Yaskawa INFORM job: KRIS4(-224_-90).JBI

/JOB
//NAME KRIS4(-224_-90)
//POS
///NPOS 312,312,312,14,0,0
///TOOL 0
///POSTYPE PULSE
///PULSE
C00000=-126,-73357,-105376,18827,72039,77556
C00001=-35778,-73357,-105376,18827,72039,77556
C00002=-13505,189291,121101,6814,55937,83682
C00003=-119958,189291,121101,6814,55937,83682
C00004=-119958,189291,121101,6814,55937,83682
C00005=-119958,189291,121101,6814,104918,83682
C00006=-69507,150313,105301,6814,83622,83682
C00007=-72199,118597,79738,6814,89727,83682
C00008=14837,117754,79738,6814,55937,83682
C00009=44504,100666,44561,7265,69044,83737
C00010=106120,216,-72664,1265,72875,87293
C00011=133015,-103640,-65816,-3996,83698,82063
C00012=132086,-97485,-64003,-4135,58701,800
C00013=149065,-104779,-51399,7594,43822,5087
C00014=150289,-91952,-48932,6393,56924,6348
C00015=150393,-90903,-46944,6418,56235,6345
C00016=150312,-91064,-47459,6419,56476,6331
C00017=149346,-88536,-46306,6590,57139,6001
C00018=150281,-91600,-48374,6405,56765,6336
C00019=170298,-72142,-39060,11518,57888,13007
C00020=170167,-71928,-38964,11546,57956,12963
C00021=170167,-71173,-37488,11610,57441,12905
C00022=170167,-71393,-37919,11591,57591,12921
C00023=169145,-69698,-37147,11804,58123,12578
C00024=170288,-72356,-39514,11498,58052,13018
C00025=137447,-116054,-63762,19682,56909,-112
C00026=108026,-108792,-54867,-4103,57296,-6110
C00027=81416,-94598,-46445,-196,58741,-15925
C00028=81757,-93684,-45677,-246,58738,-15800
C00029=81757,-92858,-44382,-247,58365,-15799
C00030=81757,-93619,-45575,-246,58708,-15800
C00031=82768,-91970,-45027,-393,59221,-15429
C00032=81930,-94457,-46518,-272,58858,-15736
C00033=128580,-105651,-52299,-6719,58617,1362
C00034=130033,-102824,-49114,-6921,58227,1914
C00035=130033,-101283,-46878,-6964,57648,1951
C00036=130033,-101721,-47515,-6952,57813,1940
C00037=129738,-99854,-46987,-6872,58421,1793
C00038=130056,-102692,-48758,-6935,58079,1930
C00039=106734,-120076,-67764,-3834,59373,-6657
C00040=106734,-120076,-67764,-3834,76101,-81400
C00041=85493,-101158,-51309,-10056,72841,-87538
C00042=85426,-99920,-49312,-10091,72250,-87511
C00043=85426,-98477,-47146,-10119,71667,-87460
C00044=85426,-98764,-47576,-10113,71783,-87469
C00045=84550,-100156,-47986,-10204,71224,-87714
C00046=85920,-99324,-49419,-10033,72673,-87380
C00047=152431,-100504,-49770,-2471,77391,-65939
C00048=152805,-100536,-48996,-2423,76908,-65809
C00049=152805,-99353,-47240,-2427,76436,-65801
C00050=152805,-99697,-47754,-2425,76574,-65803
C00051=153892,-101565,-48290,-2277,75972,-65442
C00052=152767,-100966,-49728,-2425,77135,-65826
C00053=175766,-86349,-42944,18121,68088,-61743
C00054=175951,-86348,-42668,18137,67889,-61707
C00055=175951,-85124,-40623,18213,67291,-61803
C00056=175951,-85392,-41070,18196,67421,-61782
C00057=177474,-87024,-41664,18224,66648,-61355
C00058=175558,-86298,-43164,18103,68288,-61786
C00059=175558,-91829,-52585,17786,71106,-61349
C00060=197698,-109667,-58160,17366,61060,-54816
C00061=219000,-104945,-43712,24315,53908,-49637
C00062=231055,-104193,-38505,23952,48237,-46148
C00063=233659,-103437,-37306,23712,47268,-45306
C00064=233659,-102004,-35373,23879,46852,-45418
C00065=233659,-102412,-35924,23830,46971,-45386
C00066=237043,-102549,-35954,23321,46092,-44173
C00067=233629,-103481,-37368,23709,47288,-45313
C00068=215461,-127400,-43893,16870,58722,-48272
C00069=218544,-127186,-42626,17459,57581,-47480
C00070=218544,-125569,-40789,17514,57295,-47527
C00071=220330,-126171,-41362,17770,57042,-47002
C00072=227145,-126469,-41362,18757,55731,-45038
C00073=215464,-127169,-42828,16963,58209,-48354
C00074=177088,-126078,-40365,8704,67148,-58850
C00075=153631,-128510,-40310,2158,67069,-65285
C00076=154429,-128614,-40154,2389,66903,-65072
C00077=154429,-127009,-38360,2393,66624,-65076
C00078=154429,-127497,-38907,2392,66709,-65074
C00079=160472,-128938,-38826,4148,65740,-63473
C00080=156013,-128640,-39995,2844,66753,-64645
C00081=192579,-111155,-68057,11776,89768,-52211
C00082=192579,-150013,-128024,12422,106350,-50582
C00083=192579,-150013,-128024,12422,106350,-50582
C00084=146460,-104346,-58758,87,67702,-67205
C00085=142478,-76043,-30573,-21964,63223,-64301
C00086=140672,-66044,-21918,-20034,66227,-65754
C00087=140672,-65153,-20362,-20107,65757,-65668
C00088=140672,-65445,-20871,-20083,65909,-65696
C00089=141036,-66851,-21501,-20135,65677,-65523
C00090=140672,-66975,-23548,-19959,66721,-65841
C00091=152208,-64015,-24131,4423,60929,-65240
C00092=152310,-63243,-22366,4438,60237,-65228
C00093=152310,-62511,-21042,4457,59798,-65245
C00094=152310,-62815,-21590,4449,59978,-65238
C00095=152877,-64252,-22264,4382,59627,-65043
C00096=152310,-63427,-22700,4433,60345,-65224
C00097=165385,-47284,-4207,31110,46159,-66957
C00098=165600,-47601,-4286,31106,45987,-66914
C00099=165600,-46737,-2733,31361,45549,-67081
C00100=165600,-47131,-3441,31243,45749,-67005
C00101=166254,-48297,-4074,31163,45344,-66829
C00102=165393,-47522,-4616,31042,46268,-66913
C00103=159093,-40722,392,34170,55600,-67527
C00104=164207,-35275,5586,37104,52652,-66901
C00105=150105,-51391,-6646,37971,54466,-72302
C00106=160171,-66075,-30313,2176,67510,-69492
C00107=161226,-57856,-21857,1152,65004,-69036
C00108=161820,-56153,-18823,1098,63999,-68834
C00109=152948,-61625,-21548,2027,63029,-72005
C00110=152825,-64029,-24982,2024,63909,-72032
C00111=134056,-67322,-25852,-10196,66056,-78379
C00112=163216,-54448,-8591,-32623,76134,-65479
C00113=160229,-46098,-3230,-29804,80491,-68345
C00114=158451,-47284,-3883,-30173,79720,-68790
C00115=151927,-50958,-5849,-31450,76927,-70423
C00116=133676,-75568,-30882,-10874,62812,-78150
C00117=160835,-97860,-53381,-12033,68838,-69115
C00118=160835,-137865,-129483,-11388,94610,-71530
C00119=160835,-137865,-129483,-11388,94610,-71530
C00120=156474,-127565,-44757,2910,70220,-64434
C00121=182735,-127588,-36879,6458,67666,-54620
C00122=93853,-129558,-36709,-20996,60624,-77534
C00123=154263,-130476,-42112,-2655,69883,-62096
C00124=171605,-138664,-45039,640,62750,-56909
C00125=200673,-127969,-43722,7924,66337,-48717
C00126=199485,-124610,-40058,7659,65901,-49084
C00127=154854,-130863,-40060,-3943,63519,-61415
C00128=142889,-132361,-46546,-6897,66121,-64856
C00129=228263,-110324,-43358,23728,50162,-46686
C00130=234831,-107572,-40199,23168,48067,-44517
C00131=236443,-96869,-37709,21687,51363,-43058
C00132=226552,-115005,-54629,22549,54767,-46269
C00133=203481,-118873,-57487,18716,57337,-53342
C00134=208530,-112813,-51521,18479,55775,-51715
C00135=215259,-101474,-48621,17081,58299,-48731
C00136=205976,-112243,-55103,18172,58669,-52173
C00137=201958,-123065,-58725,3253,73839,-54936
C00138=197661,-129040,-56396,6313,64525,-57421
C00139=175928,-137233,-57000,3673,61831,-64313
C00140=171824,-140203,-61595,3068,63271,-65534
C00141=141766,-147898,-61645,-3344,56480,-74079
C00142=133776,-141760,-57056,-3252,60087,-76917
C00143=117425,-137681,-55374,-11246,62568,-80588
C00144=164064,-147455,-64185,-5609,61717,-65893
C00145=164064,-147455,-64185,-5609,61717,-65893
C00146=130860,-150279,-64151,6173,30547,11978
C00147=181055,-130986,-61566,-17152,51608,35195
C00148=182532,-124800,-57711,-17116,52650,35581
C00149=83593,-132502,-58869,6067,41588,-3855
C00150=101126,-133718,-57710,-9309,38222,6255
C00151=129711,-151516,-73375,-17379,42716,18129
C00152=134581,-137990,-74595,25751,56070,-1389
C00153=110654,-139179,-74777,26363,62443,-9081
C00154=121652,-127479,-66506,26214,60123,-5457
C00155=183969,-104449,-60936,13894,52742,18216
C00156=171621,-128341,-75090,18129,51623,12881
C00157=119711,-181360,-121572,24950,66300,-4723
C00158=119711,-181360,-121572,24950,66300,-4723
C00159=119711,-181360,-135603,24950,39029,-4723
C00160=119711,-181360,-135603,24950,39029,-4723
C00161=67118,-136665,-130676,31892,63753,5674
C00162=38158,-160025,-136084,39080,61805,7690
C00163=9060,-155984,-136090,36075,61852,27249
C00164=9060,-155984,-136090,36075,61852,27249
C00165=-35778,-73357,-105376,18827,72039,77556
C00166=-35778,-73357,-105376,18827,72039,77556
C00167=-121972,-60692,-66036,23906,48760,72917
C00168=-121972,-63565,-66036,13351,77444,72917
C00169=-114761,-44204,-50669,11461,76826,75375
C00170=-114807,-42889,-47501,11529,75582,75243
C00171=-114807,-42796,-46589,11554,75077,75195
C00172=-114807,-42822,-46844,11546,75217,75208
C00173=-114733,-44587,-47920,11539,74967,75210
C00174=-114807,-42889,-47501,11529,75582,75243
C00175=-106693,-40989,-47922,-8584,79047,76853
C00176=-106712,-40732,-46990,-8589,78608,76878
C00177=-106712,-40651,-45975,-8604,78031,76918
C00178=-106712,-40674,-46241,-8599,78181,76908
C00179=-106551,-42339,-47274,-8643,77981,76977
C00180=-106693,-40989,-47922,-8584,79047,76853
C00181=-119731,-42339,-42353,-28777,73600,71789
C00182=-120080,-41537,-40336,-28806,72749,71870
C00183=-120080,-41293,-39100,-28897,72189,72014
C00184=-120080,-41335,-39305,-28882,72281,71990
C00185=-120073,-43216,-40463,-28920,72059,72050
C00186=-120080,-41537,-40336,-28806,72749,71870
C00187=-101589,-42073,-44271,-32201,81327,76893
C00188=-104782,-94542,-85411,-8339,74693,77861
C00189=-98731,-154827,-131308,-9878,72678,80158
C00190=-98731,-154827,-131308,-9878,72678,80158
C00191=-98731,-154827,-131308,-9878,72678,80158
C00192=-141095,-137804,-121947,4358,90462,65341
C00193=-171917,-153174,-112370,-11397,78411,54227
C00194=-199110,-110397,-63847,-11158,69278,59316
C00195=-199661,-105459,-60576,-13729,71348,59282
C00196=-199661,-104714,-59434,-13753,71034,59321
C00197=-199661,-104881,-59692,-13747,71104,59313
C00198=-201697,-105978,-60019,-13785,70422,58683
C00199=-199661,-105459,-60576,-13729,71348,59282
C00200=-123960,-138876,-68675,-7989,69585,84604
C00201=-124072,-138705,-67366,-8043,68864,84619
C00202=-124072,-137612,-66165,-8049,68688,84634
C00203=-124072,-137824,-66399,-8047,68723,84632
C00204=-124282,-139731,-66590,-8126,67850,84627
C00205=-124072,-138655,-67314,-8040,68857,84622
C00206=-114984,-139242,-68510,12959,69151,83072
C00207=-114827,-138670,-67011,13034,68516,83052
C00208=-114827,-136931,-65095,13059,68238,83020
C00209=-114827,-137199,-65392,13055,68282,83025
C00210=-114467,-139013,-65570,13183,67430,83044
C00211=-114827,-138670,-67011,13034,68516,83052
C00212=-133085,-142772,-85485,9589,79895,78262
C00213=-119908,-107051,-70579,11526,87272,83253
C00214=-119905,-107270,-70562,11527,87152,83243
C00215=-119905,-106417,-69135,11528,86722,83203
C00216=-119905,-106577,-69401,11528,86804,83211
C00217=-119887,-108279,-69933,11533,86265,83166
C00218=-119905,-107341,-70681,11527,87191,83247
C00219=-147950,-101609,-70952,-8097,88078,75282
C00220=-148936,-101577,-69519,-8210,87121,75014
C00221=-148936,-100979,-68423,-8210,86757,75037
C00222=-148936,-101159,-68752,-8210,86867,75032
C00223=-149395,-102566,-69230,-8263,86398,74908
C00224=-148936,-101830,-69986,-8210,87277,75005
C00225=-165354,-89650,-65481,-16319,85072,70011
C00226=-165779,-89873,-64407,-16347,84242,69973
C00227=-165779,-89214,-62991,-16359,83730,70041
C00228=-165779,-89312,-63202,-16357,83805,70031
C00229=-166355,-90439,-63644,-16386,83393,69883
C00230=-165632,-89756,-64683,-16338,84492,69992
C00231=-143601,-106428,-78314,-14904,88558,77172
C00232=-127839,-150907,-89343,-18520,59767,2936
C00233=-132953,-138286,-79588,-18019,59168,1112
C00234=-137115,-133470,-77672,-17386,59565,-529
C00235=-137115,-131953,-75830,-17447,59223,-475
C00236=-137115,-132842,-76915,-17411,59423,-507
C00237=-136304,-129881,-76308,-17304,60683,-404
C00238=-137115,-133253,-77414,-17394,59515,-521
C00239=-181699,-110020,-71549,-8619,60587,-17610
C00240=-181630,-109868,-71398,-8637,60579,-17583
C00241=-181630,-109061,-70095,-8670,60195,-17555
C00242=-181630,-109567,-70911,-8650,60436,-17574
C00243=-179495,-107200,-70173,-9064,61418,-16842
C00244=-181374,-109783,-71626,-8682,60786,-17501
C00245=-138549,-156108,-92608,-17680,56945,-638
C00246=-92857,-152389,-93170,1138,51221,11865
C00247=-89241,-137374,-84375,135,53495,13313
C00248=-89241,-137236,-84209,135,53464,13313
C00249=-89241,-136248,-83020,135,53240,13313
C00250=-89241,-136629,-83479,135,53327,13313
C00251=-90422,-134246,-82978,442,54247,12852
C00252=-88987,-137859,-84464,69,53301,13413
C00253=-151501,-140988,-86034,14129,58291,-10466
C00254=-150678,-138310,-84494,13941,58574,-10114
C00255=-150678,-137164,-83136,13977,58332,-10146
C00256=-150678,-137515,-83554,13966,58407,-10136
C00257=-149186,-134345,-82896,13563,59357,-9449
C00258=-151128,-139683,-85226,14047,58399,-10308
C00259=-154150,-131986,-81973,14219,60800,-11137
C00260=-88152,-132772,-82145,-148,54492,13740
C00261=-103700,-131599,-81415,11358,56317,183
C00262=-119170,-146244,-89248,14851,56054,-5885
C00263=-129919,-160370,-92966,-12704,53201,3154
C00264=-134642,-143084,-81504,-11683,54346,1201
C00265=-146256,-142714,-76617,-8488,45375,-2851
C00266=-190967,-116324,-69611,1501,49612,-20855
C00267=-164928,-143381,-78407,-9170,42235,-9240
C00268=-155273,-152427,-83467,-13136,41921,-4825
C00269=-158141,-110882,-79211,-11782,79402,69500
C00270=-156021,-110302,-75029,-11867,77473,70419
C00271=-164693,-106825,-70970,-11824,75528,67599
C00272=-175106,-97531,-67666,-11410,76738,63853
C00273=-131080,-121620,-80305,-3109,79327,78003
C00274=-136811,-120114,-75832,127,77816,75713
C00275=-120666,-121905,-76299,1170,77058,81080
C00276=-118816,-123903,-80121,1281,78355,81709
C00277=-109990,-123163,-79929,1817,78452,84652
C00278=-122003,-121691,-75603,8260,77024,79739
C00279=-127593,-119006,-72089,19029,78419,76519
C00280=-135969,-121502,-76764,18008,81762,74135
C00281=-157702,-146234,-81795,15058,76702,66164
C00282=-157352,-138799,-66788,13808,73912,66272
C00283=-167304,-136290,-63149,11542,74320,63270
C00284=-135907,-141176,-63619,18589,67249,72053
C00285=-148278,-138995,-66659,15795,72315,68901
C00286=-146781,-141799,-67483,-9190,63470,73790
C00287=-172222,-135689,-66769,-11071,63352,65466
C00288=-167439,-135845,-70174,-10586,65898,66819
C00289=-192902,-115042,-63146,-20265,60680,60371
C00290=-199703,-112368,-59358,-19763,58226,58217
C00291=-207207,-100813,-56084,-18051,60307,54942
C00292=-170801,-131743,-76226,-21430,65470,67743
C00293=-164740,-137810,-91614,-20635,72894,68588
C00294=-164740,-137810,-91614,-20635,72894,68588
C00295=-149447,-191890,-120181,-21381,67024,75156
C00296=-149584,-192173,-120256,-21405,66899,75131
C00297=-149584,-192173,-120256,-21405,66899,75131
C00298=-114761,-44204,-50669,11461,76826,75375
C00299=-117144,-39713,-45211,12000,78898,74743
C00300=-110396,-38535,-44464,10422,78117,77015
C00301=-114060,-50823,-52718,11111,71580,75110
C00302=-124826,-51246,-53710,-3634,72889,70409
C00303=-126627,-37483,-45033,-3511,81308,69522
C00304=-133904,-35632,-43787,-1986,81245,67064
C00305=-133954,-36259,-45628,-1970,82055,67034
C00306=-135284,-28260,-32637,-27547,76219,65313
C00307=-136156,-27594,-30758,-27439,75206,65218
C00308=-139816,-25285,-26607,-31214,71734,64504
C00309=-131832,-52683,-49405,-33204,65462,69826
C00310=-109380,-75662,-60137,-33198,63885,64520
C00311=-9054,-143647,-113334,5954,77551,79151
BC00000=192652,674564,1075172
BC00001=85490,674564,1075172
BC00002=85490,674564,1075172
BC00003=388274,674564,1075172
BC00004=388274,1057170,1075172
BC00005=388274,1057170,1075172
BC00006=266797,1098418,1075172
BC00007=245359,1165153,1075172
BC00008=171901,1306919,981729
BC00009=145084,1358673,1075172
BC00010=282424,1358673,1075172
BC00011=324887,1177345,1075172
BC00012=324887,1177345,1033512
BC00013=324887,1177345,1033512
BC00014=324887,1177345,1033512
BC00015=324887,1177345,1033512
BC00016=324887,1177345,1033512
BC00017=324887,1177345,1033512
BC00018=324887,1177345,1033512
BC00019=324887,1177345,1033512
BC00020=324887,1177345,1033512
BC00021=324887,1177345,1033512
BC00022=324887,1177345,1033512
BC00023=324887,1177345,1033512
BC00024=324887,1177345,1033512
BC00025=324887,1177345,1033512
BC00026=324887,1177345,1033512
BC00027=324887,1177345,1033512
BC00028=324887,1177345,1033512
BC00029=324887,1177345,1033512
BC00030=324887,1177345,1033512
BC00031=324887,1177345,1033512
BC00032=324887,1177345,1033512
BC00033=324887,1177345,1033512
BC00034=324887,1177345,1033512
BC00035=324887,1177345,1033512
BC00036=324887,1177345,1033512
BC00037=324887,1177345,1033512
BC00038=324887,1177345,1033512
BC00039=324887,1177345,1033512
BC00040=324887,1147445,1033512
BC00041=324887,1147445,1033512
BC00042=324887,1147445,1033512
BC00043=324887,1147445,1033512
BC00044=324887,1147445,1033512
BC00045=324887,1147445,1033512
BC00046=324887,1147445,1033512
BC00047=324887,1147445,1033512
BC00048=324887,1147445,1033512
BC00049=324887,1147445,1033512
BC00050=324887,1147445,1033512
BC00051=324887,1147445,1033512
BC00052=324887,1147445,1033512
BC00053=324887,1147445,1033512
BC00054=324887,1147445,1033512
BC00055=324887,1147445,1033512
BC00056=324887,1147445,1033512
BC00057=324887,1147445,1033512
BC00058=324887,1147445,1033512
BC00059=324887,1147445,1033512
BC00060=324887,1147445,1033512
BC00061=324887,1119707,1033512
BC00062=324887,1119707,1033512
BC00063=324887,1119707,1033512
BC00064=324887,1119707,1033512
BC00065=324887,1119707,1033512
BC00066=324887,1119707,1033512
BC00067=324887,1119707,1033512
BC00068=324887,1119707,1033512
BC00069=324887,1119707,1033512
BC00070=324887,1119707,1033512
BC00071=324887,1119707,1033512
BC00072=324887,1119707,1033512
BC00073=324887,1119707,1033512
BC00074=346918,1122350,1033512
BC00075=365620,1122350,1033512
BC00076=365620,1122350,1033512
BC00077=365620,1122350,1033512
BC00078=365620,1122350,1033512
BC00079=365620,1122350,1033512
BC00080=365620,1122350,1033512
BC00081=365620,1122350,1033512
BC00082=365620,1122350,1033512
BC00083=365620,1290426,1033512
BC00084=365620,1290426,1028316
BC00085=365620,1290426,1028316
BC00086=365620,1290426,1028316
BC00087=365620,1290426,1028316
BC00088=365620,1290426,1028316
BC00089=365620,1290426,1028316
BC00090=365620,1290426,1028316
BC00091=365620,1290426,1028316
BC00092=365620,1290426,1028316
BC00093=365620,1290426,1028316
BC00094=365620,1290426,1028316
BC00095=365620,1290426,1028316
BC00096=365620,1290426,1028316
BC00097=365620,1290426,1028316
BC00098=365620,1290426,1028316
BC00099=365620,1290426,1028316
BC00100=365620,1290426,1028316
BC00101=365620,1290426,1028316
BC00102=365620,1290426,1028316
BC00103=365620,1290426,1028316
BC00104=365620,1290426,1028316
BC00105=365620,1290426,1028316
BC00106=365620,1290426,1028316
BC00107=365620,1290426,1028316
BC00108=365620,1290426,1028316
BC00109=365620,1290426,1028316
BC00110=365620,1290426,1028316
BC00111=365620,1290426,1028316
BC00112=365620,1290426,1028316
BC00113=365620,1290426,1028316
BC00114=365620,1290426,1028316
BC00115=365620,1290426,1028316
BC00116=365620,1290426,1028316
BC00117=365620,1290426,1028316
BC00118=365620,1290426,1028316
BC00119=365620,1203984,1028316
BC00120=365620,1122350,1033512
BC00121=354696,1118911,1033512
BC00122=354696,1118911,1033512
BC00123=354696,1118911,1033512
BC00124=289412,1118911,1033512
BC00125=299099,1130329,1033512
BC00126=299099,1130329,1033512
BC00127=299099,1130329,1033512
BC00128=299099,1130329,1033512
BC00129=323037,1120469,1018827
BC00130=323037,1120469,1018827
BC00131=323037,1120469,1018827
BC00132=323037,1120469,1018827
BC00133=323037,1103765,1018827
BC00134=323037,1103765,1018827
BC00135=323037,1103765,1018827
BC00136=323037,1103765,1018827
BC00137=323037,1103765,1018827
BC00138=323037,1103765,1018827
BC00139=323037,1103765,1018827
BC00140=323037,1103765,1018827
BC00141=359327,1103765,1018827
BC00142=359327,1103765,1018827
BC00143=359327,1103765,1018827
BC00144=359327,1103765,1018827
BC00145=320666,1103765,1061735
BC00146=320666,1151385,1061735
BC00147=348115,1151385,988526
BC00148=348115,1151385,988526
BC00149=348115,1151385,988526
BC00150=348115,1151385,988526
BC00151=348115,1151385,988526
BC00152=348115,1151385,988526
BC00153=317563,1137817,963781
BC00154=317563,1137817,963781
BC00155=317563,1137817,963781
BC00156=317563,1137817,963781
BC00157=317563,1137817,963781
BC00158=357256,1203577,1061822
BC00159=340361,1234496,1068927
BC00160=340361,1313599,1068927
BC00161=331783,1191875,1070117
BC00162=326822,1083331,1070805
BC00163=344400,890386,1072234
BC00164=344400,743708,1072234
BC00165=295326,674564,1075172
BC00166=295326,676593,1075172
BC00167=295326,676846,813323
BC00168=336009,760791,731248
BC00169=336009,760791,731248
BC00170=336009,760791,731248
BC00171=336009,760791,731248
BC00172=336009,760791,731248
BC00173=336009,760791,731248
BC00174=336009,760791,731248
BC00175=292309,760791,731248
BC00176=292309,760791,731248
BC00177=292309,760791,731248
BC00178=292309,760791,731248
BC00179=292309,760791,731248
BC00180=292309,760791,731248
BC00181=292309,760791,731248
BC00182=292309,760791,731248
BC00183=292309,760791,731248
BC00184=292309,760791,731248
BC00185=292309,760791,731248
BC00186=292309,760791,731248
BC00187=292309,760791,731248
BC00188=292309,760791,731248
BC00189=292309,760791,979870
BC00190=314389,897937,979870
BC00191=314389,914237,695700
BC00192=349616,923854,695700
BC00193=349616,946341,695700
BC00194=318497,960445,891334
BC00195=318497,960445,891334
BC00196=318497,960445,891334
BC00197=318497,960445,891334
BC00198=318497,960445,891334
BC00199=318497,960445,891334
BC00200=318497,960445,891334
BC00201=318497,960445,891334
BC00202=318497,960445,891334
BC00203=318497,960445,891334
BC00204=318497,960445,891334
BC00205=318497,960445,891334
BC00206=348006,960445,891333
BC00207=348006,960445,891333
BC00208=348006,960445,891333
BC00209=348006,960445,891333
BC00210=348006,960445,891333
BC00211=348006,960445,891333
BC00212=348006,960445,891333
BC00213=348006,960445,891333
BC00214=348006,960445,891333
BC00215=348006,960445,891333
BC00216=348006,960445,891333
BC00217=348006,960445,891333
BC00218=348006,960445,891333
BC00219=348006,960445,891333
BC00220=348006,960445,891333
BC00221=348006,960445,891333
BC00222=348006,960445,891333
BC00223=348006,960445,891333
BC00224=348006,960445,891333
BC00225=317395,960445,891333
BC00226=317395,960445,891333
BC00227=317395,960445,891333
BC00228=317395,960445,891333
BC00229=317395,960445,891333
BC00230=317395,960445,891333
BC00231=317395,960445,891333
BC00232=317395,960445,891333
BC00233=317395,960445,891333
BC00234=317395,960445,891333
BC00235=317395,960445,891333
BC00236=317395,960445,891333
BC00237=317395,960445,891333
BC00238=317395,960445,891333
BC00239=317395,960445,891333
BC00240=317395,960445,891333
BC00241=317395,960445,891333
BC00242=317395,960445,891333
BC00243=317395,960445,891333
BC00244=317395,960445,891333
BC00245=317395,960445,891333
BC00246=339742,960445,891333
BC00247=339741,960446,891330
BC00248=339741,960446,891330
BC00249=339741,960446,891330
BC00250=339741,960446,891330
BC00251=339741,960446,891330
BC00252=339741,960446,891330
BC00253=339741,960446,891330
BC00254=339741,960446,891330
BC00255=339741,960446,891330
BC00256=339741,960446,891330
BC00257=339741,960446,891330
BC00258=339741,960446,891330
BC00259=339741,960446,891330
BC00260=339741,960446,891330
BC00261=339741,960446,891330
BC00262=339741,960446,891330
BC00263=310327,960446,891330
BC00264=310327,960446,891330
BC00265=310327,960446,891330
BC00266=310327,960446,891330
BC00267=310327,960446,891330
BC00268=310327,960446,891330
BC00269=310327,960446,891330
BC00270=310327,960446,891330
BC00271=310327,960446,891330
BC00272=310327,960446,891330
BC00273=310327,960446,891330
BC00274=310327,960446,891330
BC00275=310327,960446,891326
BC00276=310327,960446,891326
BC00277=351201,960446,891326
BC00278=351201,960446,891326
BC00279=351201,960446,891326
BC00280=351201,960446,891326
BC00281=351201,960446,891326
BC00282=351201,960446,891326
BC00283=351201,960446,891326
BC00284=351201,960446,891326
BC00285=351201,960446,891326
BC00286=335367,960446,891326
BC00287=335367,960446,891326
BC00288=335367,960446,891326
BC00289=335367,960446,891326
BC00290=335367,960446,891326
BC00291=335367,960446,891326
BC00292=335367,960446,891326
BC00293=335367,960446,891326
BC00294=352748,960446,1069813
BC00295=352748,960446,1069813
BC00296=352748,842200,1069813
BC00297=352748,842200,743331
BC00298=336009,760791,731248
BC00299=336010,760791,731247
BC00300=336010,760792,731244
BC00301=336010,760791,731247
BC00302=336010,760791,731247
BC00303=336010,760791,731247
BC00304=336010,760791,731247
BC00305=336010,760791,731247
BC00306=336010,760791,731247
BC00307=336010,760791,731247
BC00308=336010,760791,731247
BC00309=336010,760791,731247
BC00310=361481,703019,979319
BC00311=361481,673970,979319
EC00000=-1986524,-556476
EC00001=-1986524,-556476
EC00002=-1986524,-556476
EC00003=-1986524,-556476
EC00004=-1986524,-556476
EC00005=-1986524,-556476
EC00006=-1986524,-556476
EC00007=-1986524,-556476
EC00008=-1986524,-556476
EC00009=-1986524,-556476
EC00010=-1986524,-556476
EC00011=-1986524,-556476
EC00012=-1986524,-556476
EC00013=-1986524,-556476
EC00014=-1986524,-556476
EC00015=-1986524,-556476
EC00016=-1986524,-556476
EC00017=-1986524,-556476
EC00018=-1986524,-556476
EC00019=-1986524,-556476
EC00020=-1986524,-556476
EC00021=-1986524,-556476
EC00022=-1986524,-556476
EC00023=-1986524,-556476
EC00024=-1986524,-556476
EC00025=-1986524,-556476
EC00026=-1986524,-556476
EC00027=-1986524,-556476
EC00028=-1986524,-556476
EC00029=-1986524,-556476
EC00030=-1986524,-556476
EC00031=-1986524,-556476
EC00032=-1986524,-556476
EC00033=-1986524,-556476
EC00034=-1986524,-556476
EC00035=-1986524,-556476
EC00036=-1986524,-556476
EC00037=-1986524,-556476
EC00038=-1986524,-556476
EC00039=-1986524,-556476
EC00040=-1986524,-556476
EC00041=-1986524,-556476
EC00042=-1986524,-556476
EC00043=-1986524,-556476
EC00044=-1986524,-556476
EC00045=-1986524,-556476
EC00046=-1986524,-556476
EC00047=-1986524,-556476
EC00048=-1986524,-556476
EC00049=-1986524,-556476
EC00050=-1986524,-556476
EC00051=-1986524,-556476
EC00052=-1986524,-556476
EC00053=-1986524,-556476
EC00054=-1986524,-556476
EC00055=-1986524,-556476
EC00056=-1986524,-556476
EC00057=-1986524,-556476
EC00058=-1986524,-556476
EC00059=-1986524,-556476
EC00060=-1986524,-556476
EC00061=-1986524,-556476
EC00062=-1986524,-556476
EC00063=-1986524,-556476
EC00064=-1986524,-556476
EC00065=-1986524,-556476
EC00066=-1986524,-556476
EC00067=-1986524,-556476
EC00068=-1986524,-556476
EC00069=-1986524,-556476
EC00070=-1986524,-556476
EC00071=-1986524,-556476
EC00072=-1986524,-556476
EC00073=-1986524,-556476
EC00074=-1986524,-556476
EC00075=-1986524,-556476
EC00076=-1986524,-556476
EC00077=-1986524,-556476
EC00078=-1986524,-556476
EC00079=-1986524,-556476
EC00080=-1986524,-556476
EC00081=-1986524,-556476
EC00082=-1986524,-556476
EC00083=-1986524,-556476
EC00084=-1986525,-556476
EC00085=-1986525,-556476
EC00086=-1986525,-556476
EC00087=-1986525,-556476
EC00088=-1986525,-556476
EC00089=-1986525,-556476
EC00090=-1986525,-556476
EC00091=-1986525,-556476
EC00092=-1986525,-556476
EC00093=-1986525,-556476
EC00094=-1986525,-556476
EC00095=-1986525,-556476
EC00096=-1986525,-556476
EC00097=-1986525,-556476
EC00098=-1986525,-556476
EC00099=-1986525,-556476
EC00100=-1986525,-556476
EC00101=-1986525,-556476
EC00102=-1986525,-556476
EC00103=-1986525,-556476
EC00104=-1986525,-556476
EC00105=-1986525,-556476
EC00106=-1986525,-556476
EC00107=-1986525,-556476
EC00108=-1986525,-556476
EC00109=-1986525,-556476
EC00110=-1986525,-556476
EC00111=-1986525,-556476
EC00112=-1986525,-556476
EC00113=-1986525,-556476
EC00114=-1986525,-556476
EC00115=-1986525,-556476
EC00116=-1986525,-556476
EC00117=-1986525,-556476
EC00118=-1986525,-556476
EC00119=-1986525,-556476
EC00120=-1986524,-556476
EC00121=-1986524,-556476
EC00122=-1986524,-556476
EC00123=-1986524,-556476
EC00124=-1986524,-556476
EC00125=-1986524,-556476
EC00126=-1986524,-556476
EC00127=-1986524,-556476
EC00128=-1986524,-556476
EC00129=-1986524,-556476
EC00130=-1986524,-556476
EC00131=-1986524,-556476
EC00132=-1986524,-556476
EC00133=-1986524,-556476
EC00134=-1986524,-556476
EC00135=-1986524,-556476
EC00136=-1986524,-556476
EC00137=-1986524,-556476
EC00138=-1986524,-556476
EC00139=-1986524,-556476
EC00140=-1986524,-556476
EC00141=-1986524,-556476
EC00142=-1986524,-556476
EC00143=-1986524,-556476
EC00144=-1986524,-556476
EC00145=-1986524,-556476
EC00146=-1986524,-556476
EC00147=-1986524,-556476
EC00148=-1986524,-556476
EC00149=-1986524,-556476
EC00150=-1986524,-556476
EC00151=-1986524,-556476
EC00152=-1986524,-556476
EC00153=-1986524,-556476
EC00154=-1986524,-556476
EC00155=-1986524,-556476
EC00156=-1986524,-556476
EC00157=-1986524,-556476
EC00158=-1986524,-556476
EC00159=-1986524,-556476
EC00160=-1986524,-556476
EC00161=-1924386,-453661
EC00162=-1888448,-394196
EC00163=-1813786,-270658
EC00164=-1813786,-270658
EC00165=-1660311,-16712
EC00166=-1178646,554555
EC00167=-1144025,556476
EC00168=-1144025,556476
EC00169=-1144025,556476
EC00170=-1144025,556476
EC00171=-1144025,556476
EC00172=-1144025,556476
EC00173=-1144025,556476
EC00174=-1144025,556476
EC00175=-1144025,556476
EC00176=-1144025,556476
EC00177=-1144025,556476
EC00178=-1144025,556476
EC00179=-1144025,556476
EC00180=-1144025,556476
EC00181=-1144025,556476
EC00182=-1144025,556476
EC00183=-1144025,556476
EC00184=-1144025,556476
EC00185=-1144025,556476
EC00186=-1144025,556476
EC00187=-1144025,556476
EC00188=-1144025,556476
EC00189=-1144025,556476
EC00190=-1144025,556476
EC00191=-1144025,556476
EC00192=-1144025,556476
EC00193=-1144025,556476
EC00194=-1144025,556476
EC00195=-1144025,556476
EC00196=-1144025,556476
EC00197=-1144025,556476
EC00198=-1144025,556476
EC00199=-1144025,556476
EC00200=-1144025,556476
EC00201=-1144025,556476
EC00202=-1144025,556476
EC00203=-1144025,556476
EC00204=-1144025,556476
EC00205=-1144025,556476
EC00206=-1144023,556476
EC00207=-1144023,556476
EC00208=-1144023,556476
EC00209=-1144023,556476
EC00210=-1144023,556476
EC00211=-1144023,556476
EC00212=-1144023,556476
EC00213=-1144023,556476
EC00214=-1144023,556476
EC00215=-1144023,556476
EC00216=-1144023,556476
EC00217=-1144023,556476
EC00218=-1144023,556476
EC00219=-1144023,556476
EC00220=-1144023,556476
EC00221=-1144023,556476
EC00222=-1144023,556476
EC00223=-1144023,556476
EC00224=-1144023,556476
EC00225=-1144023,556476
EC00226=-1144023,556476
EC00227=-1144023,556476
EC00228=-1144023,556476
EC00229=-1144023,556476
EC00230=-1144023,556476
EC00231=-1144023,556476
EC00232=-1144023,556476
EC00233=-1144023,556476
EC00234=-1144023,556476
EC00235=-1144023,556476
EC00236=-1144023,556476
EC00237=-1144023,556476
EC00238=-1144023,556476
EC00239=-1144023,556476
EC00240=-1144023,556476
EC00241=-1144023,556476
EC00242=-1144023,556476
EC00243=-1144023,556476
EC00244=-1144023,556476
EC00245=-1144023,556476
EC00246=-1144023,556476
EC00247=-1144020,556476
EC00248=-1144020,556476
EC00249=-1144020,556476
EC00250=-1144020,556476
EC00251=-1144020,556476
EC00252=-1144020,556476
EC00253=-1144020,556476
EC00254=-1144020,556476
EC00255=-1144020,556476
EC00256=-1144020,556476
EC00257=-1144020,556476
EC00258=-1144020,556476
EC00259=-1144019,556476
EC00260=-1144019,556476
EC00261=-1144019,556476
EC00262=-1144019,556476
EC00263=-1144019,556476
EC00264=-1144019,556476
EC00265=-1144019,556476
EC00266=-1144019,556476
EC00267=-1144019,556476
EC00268=-1144019,556476
EC00269=-1144019,556476
EC00270=-1144019,556476
EC00271=-1144019,556476
EC00272=-1144019,556476
EC00273=-1144019,556476
EC00274=-1144019,556476
EC00275=-1144018,556476
EC00276=-1144018,556476
EC00277=-1144018,556476
EC00278=-1144018,556476
EC00279=-1144018,556476
EC00280=-1144018,556476
EC00281=-1144018,556476
EC00282=-1144018,556476
EC00283=-1144018,556476
EC00284=-1144018,556476
EC00285=-1144018,556476
EC00286=-1144018,556476
EC00287=-1144018,556476
EC00288=-1144018,556476
EC00289=-1144018,556476
EC00290=-1144018,556476
EC00291=-1144018,556476
EC00292=-1144018,556476
EC00293=-1144018,556476
EC00294=-1144018,556476
EC00295=-1144018,556476
EC00296=-1144018,556476
EC00297=-1144018,556476
EC00298=-1144025,556476
EC00299=-1144023,556477
EC00300=-1144020,556477
EC00301=-1144023,556477
EC00302=-1144023,556477
EC00303=-1144023,556477
EC00304=-1144023,556477
EC00305=-1144023,556477
EC00306=-1144023,556477
EC00307=-1144023,556477
EC00308=-1144023,556477
EC00309=-1144023,556477
EC00310=-1144023,556477
EC00311=-1207380,556477
///POSTYPE BASE
///RECTAN
///RCONF 0,0,0,0,0,0,0,0,0,0,0,0,0,0,0,0,0,0,0,0,0,0,0,0
P00006=0.000,0.000,0.000,0.0000,0.0000,0.0000
P00021=-0.225,-6.128,-0.405,0.0000,0.0000,0.0000
P00022=-0.114,-0.780,3.887,0.0000,0.0000,0.0000
P00023=0.143,-0.036,0.682,0.0000,0.0000,0.0000
P00024=0.145,-0.552,1.326,0.0000,0.0000,0.0000
P00025=-2.003,0.006,0.728,0.0000,0.0000,0.0000
P00026=0.562,-0.002,-0.337,0.0000,0.0000,0.0000
P00027=-0.746,0.015,-9.096,0.0000,0.0000,0.0000
P00028=-2.237,-0.018,-7.702,0.0000,0.0000,0.0000
P00029=-2.156,-0.086,-4.681,0.0000,0.0000,0.0000
P00030=5.926,-4.294,-1.390,0.0000,0.0000,0.0000
P00031=1.853,-0.001,-1.549,0.0000,0.0000,0.0000
P00032=1.957,0.503,-7.217,0.0000,0.0000,0.0000
///RCONF 0,0,0,0,1,0,0,0,0,0,0,0,0,0,0,0,0,0,0,0,0,0,0,0
P00033=-0.123,0.612,-5.012,0.0000,0.0000,0.0000
//INST
///DATE 2025/02/07 17:09
///ATTR SC,RW
///GROUP1 RB1,BS1
///GROUP2 ST1
NOP
'300124 MUZYLO
MOVJ C00000 BC00000 VJ=100.00  +MOVJ EC00000 VJ=100.00
CALL JOB:CLEAN-R1_KM_NEW
MOVJ C00001 BC00001 VJ=100.00  +MOVJ EC00001 VJ=100.00
MOVJ C00002 BC00002 VJ=100.00  +MOVJ EC00002 VJ=100.00
MOVJ C00003 BC00003 VJ=100.00  +MOVJ EC00003 VJ=100.00
MOVJ C00004 BC00004 VJ=100.00  +MOVJ EC00004 VJ=100.00
MOVJ C00005 BC00005 VJ=100.00  +MOVJ EC00005 VJ=0.78
MOVJ C00006 BC00006 VJ=100.00  +MOVJ EC00006 VJ=100.00
MOVJ C00007 BC00007 VJ=100.00  +MOVJ EC00007 VJ=100.00
MOVJ C00008 BC00008 VJ=100.00  +MOVJ EC00008 VJ=100.00
MOVJ C00009 BC00009 VJ=100.00  +MOVJ EC00009 VJ=100.00
MOVJ C00010 BC00010 VJ=100.00  +MOVJ EC00010 VJ=100.00
MOVJ C00011 BC00011 VJ=100.00  +MOVJ EC00011 VJ=100.00
MOVJ C00012 BC00012 VJ=100.00  +MOVJ EC00012 VJ=100.00
MOVJ C00013 BC00013 VJ=100.00  +MOVJ EC00013 VJ=100.00
SMOVL C00014 BC00014 V=100.0  +MOVJ EC00014
SREFP 3 C00015 BC00015  +REFP EC00015
CALL JOB:SEARCH-R1-S13D
SET P032 P006
SFTON3D P032
SMOVL C00016 BC00016 V=100.0  +MOVJ EC00016
SREFP 3 C00017 BC00017  +REFP EC00017
CALL JOB:SEARCH-R1-S13D
SET P032 P006
SFTON3D P032
SMOVL C00018 BC00018 V=100.0  +MOVJ EC00018
SFTOF3D
SMOVL C00019 BC00019 V=333.3  +MOVJ EC00019
SMOVL C00020 BC00020 V=100.0  +MOVJ EC00020
SREFP 3 C00021 BC00021  +REFP EC00021
CALL JOB:SEARCH-R1-S13D
SET P033 P006
SFTON3D P033
SMOVL C00022 BC00022 V=100.0  +MOVJ EC00022
SREFP 3 C00023 BC00023  +REFP EC00023
CALL JOB:SEARCH-R1-S13D
SET P033 P006
SFTON3D P033
SMOVL C00024 BC00024 V=100.0  +MOVJ EC00024
SFTOF3D
SMOVL C00025 BC00025 V=333.3  +MOVJ EC00025
SMOVL C00026 BC00026 V=1000.0  +MOVJ EC00026
SMOVL C00027 BC00027 V=666.7  +MOVJ EC00027
SMOVL C00028 BC00028 V=100.0  +MOVJ EC00028
SREFP 3 C00029 BC00029  +REFP EC00029
CALL JOB:SEARCH-R1-S13D
SET P030 P006
SFTON3D P030
SMOVL C00030 BC00030 V=100.0  +MOVJ EC00030
SREFP 3 C00031 BC00031  +REFP EC00031
CALL JOB:SEARCH-R1-S13D
SET P030 P006
SFTON3D P030
SMOVL C00032 BC00032 V=100.0  +MOVJ EC00032
SFTOF3D
SMOVL C00033 BC00033 V=666.7  +MOVJ EC00033
SMOVL C00034 BC00034 V=100.0  +MOVJ EC00034
SREFP 3 C00035 BC00035  +REFP EC00035
CALL JOB:SEARCH-R1-S13D
SET P031 P006
SFTON3D P031
SMOVL C00036 BC00036 V=100.0  +MOVJ EC00036
SREFP 3 C00037 BC00037  +REFP EC00037
CALL JOB:SEARCH-R1-S13D
SET P031 P006
SFTON3D P031
SMOVL C00038 BC00038 V=100.0  +MOVJ EC00038
SFTOF3D
MOVJ C00039 BC00039 VJ=100.00  +MOVJ EC00039 VJ=100.00
MOVJ C00040 BC00040 VJ=100.00  +MOVJ EC00040 VJ=50.00
MOVJ C00041 BC00041 VJ=100.00  +MOVJ EC00041 VJ=50.00
SMOVL C00042 BC00042 V=100.0  +MOVJ EC00042
SREFP 3 C00043 BC00043  +REFP EC00043
CALL JOB:SEARCH-R1-S13D
SET P021 P006
SFTON3D P021
SMOVL C00044 BC00044 V=100.0  +MOVJ EC00044
SREFP 3 C00045 BC00045  +REFP EC00045
CALL JOB:SEARCH-R1-S13D
SET P021 P006
SFTON3D P021
SMOVL C00046 BC00046 V=100.0  +MOVJ EC00046
SFTOF3D
SMOVL C00047 BC00047 V=666.7  +MOVJ EC00047
SMOVL C00048 BC00048 V=100.0  +MOVJ EC00048
SREFP 3 C00049 BC00049  +REFP EC00049
CALL JOB:SEARCH-R1-S13D
SET P022 P006
SFTON3D P022
SMOVL C00050 BC00050 V=100.0  +MOVJ EC00050
SREFP 3 C00051 BC00051  +REFP EC00051
CALL JOB:SEARCH-R1-S13D
SET P022 P006
SFTON3D P022
SMOVL C00052 BC00052 V=100.0  +MOVJ EC00052
SFTOF3D
SMOVL C00053 BC00053 V=666.7  +MOVJ EC00053
SMOVL C00054 BC00054 V=100.0  +MOVJ EC00054
SREFP 3 C00055 BC00055  +REFP EC00055
CALL JOB:SEARCH-R1-S13D
SET P023 P006
SFTON3D P023
SMOVL C00056 BC00056 V=100.0  +MOVJ EC00056
SREFP 3 C00057 BC00057  +REFP EC00057
CALL JOB:SEARCH-R1-S13D
SET P023 P006
SFTON3D P023
SMOVL C00058 BC00058 V=100.0  +MOVJ EC00058
SFTOF3D
SMOVL C00059 BC00059 V=1000.0  +MOVJ EC00059
SMOVL C00060 BC00060 V=333.3  +MOVJ EC00060
SMOVL C00061 BC00061 V=333.3  +MOVJ EC00061
SMOVL C00062 BC00062 V=333.3  +MOVJ EC00062
SMOVL C00063 BC00063 V=100.0  +MOVJ EC00063
SREFP 3 C00064 BC00064  +REFP EC00064
CALL JOB:SEARCH-R1-S13D
SET P024 P006
SFTON3D P024
SMOVL C00065 BC00065 V=100.0  +MOVJ EC00065
SREFP 3 C00066 BC00066  +REFP EC00066
CALL JOB:SEARCH-R1-S13D
SET P024 P006
SFTON3D P024
SMOVL C00067 BC00067 V=100.0  +MOVJ EC00067
SFTOF3D
SMOVL C00068 BC00068 V=666.7  +MOVJ EC00068
SMOVL C00069 BC00069 V=100.0  +MOVJ EC00069
SREFP 3 C00070 BC00070  +REFP EC00070
CALL JOB:SEARCH-R1-S13D
SET P025 P006
SFTON3D P025
SMOVL C00071 BC00071 V=100.0  +MOVJ EC00071
SREFP 3 C00072 BC00072  +REFP EC00072
CALL JOB:SEARCH-R1-S13D
SET P025 P006
SFTON3D P025
SMOVL C00073 BC00073 V=100.0  +MOVJ EC00073
SFTOF3D
SMOVL C00074 BC00074 V=666.7  +MOVJ EC00074
SMOVL C00075 BC00075 V=166.7  +MOVJ EC00075
SMOVL C00076 BC00076 V=100.0  +MOVJ EC00076
SREFP 3 C00077 BC00077  +REFP EC00077
CALL JOB:SEARCH-R1-S13D
SET P026 P006
SFTON3D P026
SMOVL C00078 BC00078 V=100.0  +MOVJ EC00078
SREFP 3 C00079 BC00079  +REFP EC00079
CALL JOB:SEARCH-R1-S13D
SET P026 P006
SFTON3D P026
SMOVL C00080 BC00080 V=100.0  +MOVJ EC00080
SFTOF3D
MOVJ C00081 BC00081 VJ=100.00  +MOVJ EC00081 VJ=50.00
MOVJ C00082 BC00082 VJ=100.00  +MOVJ EC00082 VJ=50.00
MOVJ C00083 BC00083 VJ=100.00  +MOVJ EC00083 VJ=50.00
MOVJ C00084 BC00084 VJ=100.00  +MOVJ EC00084 VJ=50.00
MOVJ C00085 BC00085 VJ=100.00  +MOVJ EC00085 VJ=50.00
SMOVL C00086 BC00086 V=166.7  +MOVJ EC00086
SREFP 3 C00087 BC00087  +REFP EC00087
CALL JOB:SEARCH-R1-S13D
SET P027 P006
SFTON3D P027
SMOVL C00088 BC00088 V=100.0  +MOVJ EC00088
SREFP 3 C00089 BC00089  +REFP EC00089
CALL JOB:SEARCH-R1-S13D
SET P027 P006
SFTON3D P027
SMOVL C00090 BC00090 V=166.7  +MOVJ EC00090
SFTOF3D
SMOVL C00091 BC00091 V=666.7  +MOVJ EC00091
SMOVL C00092 BC00092 V=100.0  +MOVJ EC00092
SREFP 3 C00093 BC00093  +REFP EC00093
CALL JOB:SEARCH-R1-S13D
SET P028 P006
SFTON3D P028
SMOVL C00094 BC00094 V=100.0  +MOVJ EC00094
SREFP 3 C00095 BC00095  +REFP EC00095
CALL JOB:SEARCH-R1-S13D
SET P028 P006
SFTON3D P028
SMOVL C00096 BC00096 V=100.0  +MOVJ EC00096
SFTOF3D
SMOVL C00097 BC00097 V=333.3  +MOVJ EC00097
SMOVL C00098 BC00098 V=100.0  +MOVJ EC00098
SREFP 3 C00099 BC00099  +REFP EC00099
CALL JOB:SEARCH-R1-S13D
SET P029 P006
SFTON3D P029
SMOVL C00100 BC00100 V=100.0  +MOVJ EC00100
SREFP 3 C00101 BC00101  +REFP EC00101
CALL JOB:SEARCH-R1-S13D
SET P029 P006
SFTON3D P029
SMOVL C00102 BC00102 V=100.0  +MOVJ EC00102
MACRO1 MJ#(0) ARGF14
'SPAWANIE 1CZ.
SMOVL C00103 BC00103 V=133.3  +MOVJ EC00103
ARCON
SMOVL C00104 BC00104 V=10.0  +MOVJ EC00104
ARCOF
SFTOF3D
SMOVL C00105 BC00105 V=250.0  +MOVJ EC00105
SMOVL C00106 BC00106 V=500.0  +MOVJ EC00106
SMOVL C00107 BC00107 V=666.7  +MOVJ EC00107
SFTON3D P028
SMOVL C00108 BC00108 V=166.7  +MOVJ EC00108
ARCON
SMOVL C00109 BC00109 V=10.0  +MOVJ EC00109
ARCOF
SFTOF3D
SMOVL C00110 BC00110 V=166.7  +MOVJ EC00110
SMOVL C00111 BC00111 V=666.7  +MOVJ EC00111
SMOVL C00112 BC00112 V=83.3  +MOVJ EC00112
SFTON3D P027
SMOVL C00113 BC00113 V=83.3 PL=0  +MOVJ EC00113
ARCON
SMOVL C00114 BC00114 V=10.0  +MOVJ EC00114
SMOVL C00115 BC00115 V=10.0  +MOVJ EC00115
ARCOF
SFTOF3D
SMOVL C00116 BC00116 V=166.7  +MOVJ EC00116
MOVJ C00117 BC00117 VJ=100.00  +MOVJ EC00117 VJ=50.00
MOVJ C00118 BC00118 VJ=100.00  +MOVJ EC00118 VJ=50.00
MOVJ C00119 BC00119 VJ=100.00  +MOVJ EC00119 VJ=100.00
MOVJ C00120 BC00120 VJ=100.00  +MOVJ EC00120 VJ=100.00
SFTON3D P026
SMOVL C00121 BC00121 V=133.3 PL=0  +MOVJ EC00121
ARCON
SMOVL C00122 BC00122 V=10.0  +MOVJ EC00122
ARCOF
SFTOF3D
SMOVL C00123 BC00123 V=166.7  +MOVJ EC00123
SMOVL C00124 BC00124 V=333.3  +MOVJ EC00124
SMOVL C00125 BC00125 V=166.7  +MOVJ EC00125
SFTON3D P025
SMOVL C00126 BC00126 V=166.7  +MOVJ EC00126
ARCON
SMOVL C00127 BC00127 V=10.0  +MOVJ EC00127
ARCOF
SFTOF3D
SMOVL C00128 BC00128 V=250.0  +MOVJ EC00128
SMOVL C00129 BC00129 V=333.3  +MOVJ EC00129
SFTON3D P024
SMOVL C00130 BC00130 V=166.7  +MOVJ EC00130
ARCON
SMOVL C00131 BC00131 V=10.0  +MOVJ EC00131
ARCOF
SFTOF3D
SMOVL C00132 BC00132 V=250.0  +MOVJ EC00132
SMOVL C00133 BC00133 V=416.7  +MOVJ EC00133
SFTON3D P023
SMOVL C00134 BC00134 V=166.7  +MOVJ EC00134
ARCON
SMOVL C00135 BC00135 V=10.0  +MOVJ EC00135
ARCOF
SFTOF3D
SMOVL C00136 BC00136 V=250.0  +MOVJ EC00136
SMOVL C00137 BC00137 V=500.0  +MOVJ EC00137
SFTON3D P022
SMOVL C00138 BC00138 V=166.7  +MOVJ EC00138
ARCON
SMOVL C00139 BC00139 V=10.0  +MOVJ EC00139
ARCOF
SFTOF3D
SMOVL C00140 BC00140 V=500.0  +MOVJ EC00140
SMOVL C00141 BC00141 V=500.0  +MOVJ EC00141
SFTON3D P021
SMOVL C00142 BC00142 V=133.3 PL=0  +MOVJ EC00142
ARCON
SMOVL C00143 BC00143 V=10.0  +MOVJ EC00143
ARCOF
SFTOF3D
SMOVL C00144 BC00144 V=333.3  +MOVJ EC00144
MOVJ C00145 BC00145 VJ=100.00  +MOVJ EC00145 VJ=100.00
MOVJ C00146 BC00146 VJ=100.00  +MOVJ EC00146 VJ=100.00
MOVJ C00147 BC00147 VJ=100.00  +MOVJ EC00147 VJ=100.00
SFTON3D P031
SMOVL C00148 BC00148 V=166.7  +MOVJ EC00148
ARCON
SFTON3D P030
SMOVL C00149 BC00149 V=10.0  +MOVJ EC00149
SMOVL C00150 BC00150 V=10.0  +MOVJ EC00150
ARCOF
SFTOF3D
SMOVL C00151 BC00151 V=250.0  +MOVJ EC00151
SMOVL C00152 BC00152 V=1000.0  +MOVJ EC00152
SMOVL C00153 BC00153 V=1000.0  +MOVJ EC00153
SFTON3D P032
SMOVL C00154 BC00154 V=166.7  +MOVJ EC00154
ARCON
SFTON3D P033
SMOVL C00155 BC00155 V=10.0  +MOVJ EC00155
ARCOF
SFTOF3D
SMOVL C00156 BC00156 V=500.0  +MOVJ EC00156
MOVJ C00157 BC00157 VJ=100.00  +MOVJ EC00157 VJ=30.00
MOVJ C00158 BC00158 VJ=100.00  +MOVJ EC00158 VJ=100.00
MOVJ C00159 BC00159 VJ=100.00  +MOVJ EC00159 VJ=100.00
MOVJ C00160 BC00160 VJ=100.00  +MOVJ EC00160 VJ=100.00
MOVJ C00161 BC00161 VJ=100.00  +MOVJ EC00161 VJ=100.00
MOVJ C00162 BC00162 VJ=100.00  +MOVJ EC00162 VJ=100.00
MOVJ C00163 BC00163 VJ=20.00  +MOVJ EC00163 VJ=100.00
MOVJ C00164 BC00164 VJ=20.00  +MOVJ EC00164 VJ=20.00
'DRUGA POZYCJA
MOVJ C00165 BC00165 VJ=100.00  +MOVJ EC00165 VJ=100.00
MOVJ C00166 BC00166 VJ=100.00  +MOVJ EC00166 VJ=100.00
CALL JOB:CLEAN-R1_KM_NEW
MOVJ C00167 BC00167 VJ=100.00  +MOVJ EC00167 VJ=100.00
MOVJ C00168 BC00168 VJ=100.00  +MOVJ EC00168 VJ=100.00
MOVJ C00169 BC00169 VJ=100.00  +MOVJ EC00169 VJ=100.00
SMOVL C00170 BC00170 V=100.0  +MOVJ EC00170
SREFP 3 C00171 BC00171  +REFP EC00171
CALL JOB:SEARCH-R1-S13D
SET P021 P006
SFTON3D P021
SMOVL C00172 BC00172 V=100.0  +MOVJ EC00172
SREFP 3 C00173 BC00173  +REFP EC00173
CALL JOB:SEARCH-R1-S13D
SET P021 P006
SFTON3D P021
SMOVL C00174 BC00174 V=100.0  +MOVJ EC00174
SFTOF3D
SMOVL C00175 BC00175 V=333.3  +MOVJ EC00175
SMOVL C00176 BC00176 V=100.0  +MOVJ EC00176
SREFP 3 C00177 BC00177  +REFP EC00177
CALL JOB:SEARCH-R1-S13D
SET P022 P006
SFTON3D P022
SMOVL C00178 BC00178 V=100.0  +MOVJ EC00178
SREFP 3 C00179 BC00179  +REFP EC00179
CALL JOB:SEARCH-R1-S13D
SET P022 P006
SFTON3D P022
SMOVL C00180 BC00180 V=100.0  +MOVJ EC00180
SFTOF3D
SMOVL C00181 BC00181 V=333.3  +MOVJ EC00181
SMOVL C00182 BC00182 V=100.0  +MOVJ EC00182
SREFP 3 C00183 BC00183  +REFP EC00183
CALL JOB:SEARCH-R1-S13D
SET P023 P006
SFTON3D P023
SMOVL C00184 BC00184 V=100.0  +MOVJ EC00184
SREFP 3 C00185 BC00185  +REFP EC00185
CALL JOB:SEARCH-R1-S13D
SET P023 P006
SFTON3D P023
SMOVL C00186 BC00186 V=100.0  +MOVJ EC00186
SFTOF3D
SMOVL C00187 BC00187 V=333.3  +MOVJ EC00187
SMOVL C00188 BC00188 V=1000.0  +MOVJ EC00188
SMOVL C00189 BC00189 V=1000.0  +MOVJ EC00189
MOVJ C00190 BC00190 VJ=100.00  +MOVJ EC00190 VJ=100.00
MOVJ C00191 BC00191 VJ=100.00  +MOVJ EC00191 VJ=100.00
MOVJ C00192 BC00192 VJ=100.00  +MOVJ EC00192 VJ=100.00
MOVJ C00193 BC00193 VJ=100.00  +MOVJ EC00193 VJ=100.00
SMOVL C00194 BC00194 V=333.3  +MOVJ EC00194
SMOVL C00195 BC00195 V=100.0  +MOVJ EC00195
SREFP 3 C00196 BC00196  +REFP EC00196
CALL JOB:SEARCH-R1-S13D
SET P024 P006
SFTON3D P024
SMOVL C00197 BC00197 V=100.0  +MOVJ EC00197
SREFP 3 C00198 BC00198  +REFP EC00198
CALL JOB:SEARCH-R1-S13D
SET P024 P006
SFTON3D P024
SMOVL C00199 BC00199 V=100.0  +MOVJ EC00199
SFTOF3D
SMOVL C00200 BC00200 V=333.3  +MOVJ EC00200
SMOVL C00201 BC00201 V=100.0  +MOVJ EC00201
SREFP 3 C00202 BC00202  +REFP EC00202
CALL JOB:SEARCH-R1-S13D
SET P025 P006
SFTON3D P025
SMOVL C00203 BC00203 V=100.0  +MOVJ EC00203
SREFP 3 C00204 BC00204  +REFP EC00204
CALL JOB:SEARCH-R1-S13D
SET P025 P006
SFTON3D P025
SMOVL C00205 BC00205 V=100.0  +MOVJ EC00205
SFTOF3D
SMOVL C00206 BC00206 V=500.0  +MOVJ EC00206
SMOVL C00207 BC00207 V=100.0  +MOVJ EC00207
SREFP 3 C00208 BC00208  +REFP EC00208
CALL JOB:SEARCH-R1-S13D
SET P026 P006
SFTON3D P026
SMOVL C00209 BC00209 V=60.0  +MOVJ EC00209
SREFP 3 C00210 BC00210  +REFP EC00210
CALL JOB:SEARCH-R1-S13D
SET P026 P006
SFTON3D P026
SMOVL C00211 BC00211 V=60.0  +MOVJ EC00211
SFTOF3D
MOVJ C00212 BC00212 VJ=100.00  +MOVJ EC00212 VJ=50.00
MOVJ C00213 BC00213 VJ=100.00  +MOVJ EC00213 VJ=50.00
SMOVL C00214 BC00214 V=100.0  +MOVJ EC00214
SREFP 3 C00215 BC00215  +REFP EC00215
CALL JOB:SEARCH-R1-S13D
SET P027 P006
SFTON3D P027
SMOVL C00216 BC00216 V=100.0  +MOVJ EC00216
SREFP 3 C00217 BC00217  +REFP EC00217
CALL JOB:SEARCH-R1-S13D
SET P027 P006
SFTON3D P027
SMOVL C00218 BC00218 V=100.0  +MOVJ EC00218
SFTOF3D
SMOVL C00219 BC00219 V=250.0  +MOVJ EC00219
SMOVL C00220 BC00220 V=100.0  +MOVJ EC00220
SREFP 3 C00221 BC00221  +REFP EC00221
CALL JOB:SEARCH-R1-S13D
SET P028 P006
SFTON3D P028
SMOVL C00222 BC00222 V=100.0  +MOVJ EC00222
SREFP 3 C00223 BC00223  +REFP EC00223
CALL JOB:SEARCH-R1-S13D
SET P028 P006
SFTON3D P028
SMOVL C00224 BC00224 V=100.0  +MOVJ EC00224
SFTOF3D
SMOVL C00225 BC00225 V=416.7  +MOVJ EC00225
SMOVL C00226 BC00226 V=10.0  +MOVJ EC00226
SREFP 3 C00227 BC00227  +REFP EC00227
CALL JOB:SEARCH-R1-S13D
SET P029 P006
SFTON3D P029
SMOVL C00228 BC00228 V=100.0  +MOVJ EC00228
SREFP 3 C00229 BC00229  +REFP EC00229
CALL JOB:SEARCH-R1-S13D
SET P029 P006
SFTON3D P029
SMOVL C00230 BC00230 V=100.0  +MOVJ EC00230
MOVJ C00231 BC00231 VJ=100.00  +MOVJ EC00231 VJ=100.00
MOVJ C00232 BC00232 VJ=100.00  +MOVJ EC00232 VJ=100.00
MOVJ C00233 BC00233 VJ=100.00  +MOVJ EC00233 VJ=100.00
SMOVL C00234 BC00234 V=10.0  +MOVJ EC00234
SREFP 3 C00235 BC00235  +REFP EC00235
CALL JOB:SEARCH-R1-S13D
SET P030 P006
SFTON3D P030
SMOVL C00236 BC00236 V=100.0  +MOVJ EC00236
SREFP 3 C00237 BC00237  +REFP EC00237
CALL JOB:SEARCH-R1-S13D
SET P030 P006
SFTON3D P030
SMOVL C00238 BC00238 V=100.0  +MOVJ EC00238
SFTOF3D
SMOVL C00239 BC00239 V=416.7  +MOVJ EC00239
SMOVL C00240 BC00240 V=100.0  +MOVJ EC00240
SREFP 3 C00241 BC00241  +REFP EC00241
CALL JOB:SEARCH-R1-S13D
SET P031 P006
SFTON3D P031
SMOVL C00242 BC00242 V=100.0  +MOVJ EC00242
SREFP 3 C00243 BC00243  +REFP EC00243
CALL JOB:SEARCH-R1-S13D
SET P031 P006
SFTON3D P031
SMOVL C00244 BC00244 V=100.0  +MOVJ EC00244
SFTOF3D
SMOVL C00245 BC00245 V=500.0  +MOVJ EC00245
SMOVL C00246 BC00246 V=1000.0  +MOVJ EC00246
SMOVL C00247 BC00247 V=500.0  +MOVJ EC00247
SMOVL C00248 BC00248 V=100.0  +MOVJ EC00248
SREFP 3 C00249 BC00249  +REFP EC00249
CALL JOB:SEARCH-R1-S13D
SET P033 P006
SFTON3D P033
SMOVL C00250 BC00250 V=100.0  +MOVJ EC00250
SREFP 3 C00251 BC00251  +REFP EC00251
CALL JOB:SEARCH-R1-S13D
SET P033 P006
SFTON3D P033
SMOVL C00252 BC00252 V=100.0  +MOVJ EC00252
SFTOF3D
SMOVL C00253 BC00253 V=416.7  +MOVJ EC00253
SMOVL C00254 BC00254 V=100.0  +MOVJ EC00254
SREFP 3 C00255 BC00255  +REFP EC00255
CALL JOB:SEARCH-R1-S13D
SET P032 P006
SFTON3D P032
SMOVL C00256 BC00256 V=100.0  +MOVJ EC00256
SREFP 3 C00257 BC00257  +REFP EC00257
CALL JOB:SEARCH-R1-S13D
SET P032 P006
SFTON3D P032
SMOVL C00258 BC00258 V=100.0  +MOVJ EC00258
MACRO1 MJ#(0) ARGF14
SMOVL C00259 BC00259 V=166.7  +MOVJ EC00259
ARCON
SFTON3D P033
SMOVL C00260 BC00260 V=9.2  +MOVJ EC00260
SMOVL C00261 BC00261 V=9.2  +MOVJ EC00261
ARCOF
SFTOF3D
SMOVL C00262 BC00262 V=416.7  +MOVJ EC00262
SMOVL C00263 BC00263 V=1000.0  +MOVJ EC00263
SMOVL C00264 BC00264 V=416.7  +MOVJ EC00264
SFTON3D P030
SMOVL C00265 BC00265 V=133.3  +MOVJ EC00265
ARCON
SFTON3D P031
SMOVL C00266 BC00266 V=8.3  +MOVJ EC00266
ARCOF
SFTOF3D
SMOVL C00267 BC00267 V=416.7  +MOVJ EC00267
MOVJ C00268 BC00268 VJ=100.00  +MOVJ EC00268 VJ=100.00
MOVJ C00269 BC00269 VJ=100.00  +MOVJ EC00269 VJ=100.00
MOVJ C00270 BC00270 VJ=100.00  +MOVJ EC00270 VJ=100.00
'BRAK POM SPR CZY OK
SFTON3D P029
SMOVL C00271 BC00271 V=133.3  +MOVJ EC00271
ARCON
MOVL C00272 BC00272 V=10.0  +MOVJ EC00272 VJ=15.00
ARCOF
SFTOF3D
MOVJ C00273 BC00273 VJ=100.00  +MOVJ EC00273 VJ=15.00
SFTON3D P028
SMOVL C00274 BC00274 V=133.3  +MOVJ EC00274
ARCON
SMOVL C00275 BC00275 V=10.0  +MOVJ EC00275
ARCOF
SFTOF3D
SMOVL C00276 BC00276 V=500.0  +MOVJ EC00276
SMOVL C00277 BC00277 V=833.3  +MOVJ EC00277
SFTON3D P027
SMOVL C00278 BC00278 V=133.3  +MOVJ EC00278
ARCON
SMOVL C00279 BC00279 V=10.0  +MOVJ EC00279
ARCOF
SFTOF3D
SMOVL C00280 BC00280 V=250.0  +MOVJ EC00280
SMOVL C00281 BC00281 V=500.0  +MOVJ EC00281
SMOVL C00282 BC00282 V=333.3  +MOVJ EC00282
SFTON3D P026
SMOVL C00283 BC00283 V=133.3  +MOVJ EC00283
ARCON
SMOVL C00284 BC00284 V=10.0  +MOVJ EC00284
ARCOF
SFTOF3D
SMOVL C00285 BC00285 V=250.0  +MOVJ EC00285
SFTON3D P025
SMOVL C00286 BC00286 V=250.0  +MOVJ EC00286
ARCON
SMOVL C00287 BC00287 V=10.0  +MOVJ EC00287
ARCOF
SFTOF3D
SMOVL C00288 BC00288 V=250.0  +MOVJ EC00288
SMOVL C00289 BC00289 V=500.0  +MOVJ EC00289
SFTON3D P024
SMOVL C00290 BC00290 V=133.3  +MOVJ EC00290
ARCON
SMOVL C00291 BC00291 V=10.0  +MOVJ EC00291
ARCOF
SMOVL C00292 BC00292 V=666.7  +MOVJ EC00292
SMOVL C00293 BC00293 V=1000.0  +MOVJ EC00293
SMOVL C00294 BC00294 V=333.3  +MOVJ EC00294
SMOVL C00295 BC00295 V=1000.0  +MOVJ EC00295
SMOVL C00296 BC00296 V=1000.0  +MOVJ EC00296
SMOVL C00297 BC00297 V=1000.0  +MOVJ EC00297
SMOVL C00298 BC00298 V=666.7  +MOVJ EC00298
SFTON3D P021
SMOVL C00299 BC00299 V=133.3  +MOVJ EC00299
ARCON
SMOVL C00300 BC00300 V=10.0  +MOVJ EC00300
ARCOF
SFTOF3D
SMOVL C00301 BC00301 V=166.7  +MOVJ EC00301
SMOVL C00302 BC00302 V=666.7  +MOVJ EC00302
SFTON3D P022
SMOVL C00303 BC00303 V=133.3  +MOVJ EC00303
ARCON
SMOVL C00304 BC00304 V=10.0  +MOVJ EC00304
ARCOF
SFTOF3D
SMOVL C00305 BC00305 V=133.3  +MOVJ EC00305
SMOVL C00306 BC00306 V=666.7  +MOVJ EC00306
SFTON3D P023
SMOVL C00307 BC00307 V=133.3  +MOVJ EC00307
ARCON
SMOVL C00308 BC00308 V=10.0  +MOVJ EC00308
ARCOF
SFTOF3D
SMOVL C00309 BC00309 V=666.7  +MOVJ EC00309
MOVJ C00310 BC00310 VJ=100.00  +MOVJ EC00310 VJ=100.00
MOVJ C00311 BC00311 VJ=100.00  +MOVJ EC00311 VJ=100.00
END
